{attribute addProperty Activity "task is running"}
FUNCTION_BLOCK fbPistonMoveTask EXTENDS TcoCore.TcoTask
VAR_INPUT
	PositionSensor : BOOL;
END_VAR
VAR_IN_OUT
	MoveToPositionSignal : BOOL;
	InverseSignal : BOOL;	
END_VAR

IF(THIS^.Execute())THEN
	THIS^.Messenger.Debug('|[[1]AttributeName]| |[AttributeActivity]|, extremity sensor not reached yet.');
	InverseSignal := FALSE;
	MoveToPositionSignal := TRUE;
	ThrowWhen(THIS^.ElapsedTime > T#5S);
	THIS^.DoneWhen(PositionSensor);
END_IF

END_FUNCTION_BLOCK

(* stored: Version 1.1.0.1
   POU fbPistonMoveTask: Id {1f1598b7-7a48-083b-213f-7881bc714afd}, SpecialFunc None *)
